// TwinCAT 3 PLC project Strings
// Title: Strings
// Company: _
// Author: Krystian Lis et al.
// ProjectVersion: 1.0.0
// Description: String ops
// ProgramVersion: 3.1.4026.9
// libraries:
//   Tc2_Standard, * (Beckhoff Automation GmbH)
//   Tc2_System, * (Beckhoff Automation GmbH)
//   Tc2_Utilities, * (Beckhoff Automation GmbH)
//   Results, * (_)
// project tree:
//   Strings/Alias/ Ch.TcDUT, Str.TcDUT
//   Strings/SymbolPath/ SymbolPath.TcPOU
//   Strings/Strb/ I_Strb.TcIO, Strb.TcPOU
//   Strings/Strf/ Strf.TcPOU
// (motion and I/O tree: see PLC project broadcast)
// real-time tasks:
//   TASK PlcTask: cycle T#10ms, priority 20, ADS port 350
//   TASK VISU_TASK: cycle T#200000us, priority 30, ADS port 351

// ---- Strings/Alias/Ch.TcDUT
TYPE Ch : STRING(1); END_TYPE

// ---- Strings/Alias/Str.TcDUT
TYPE Str : STRING(255); END_TYPE

// ---- Strings/Strb/I_Strb.TcIO
INTERFACE INTERNAL I_Strb

METHOD Append : I_Strb;
VAR_INPUT
	sToAdd		: Str;
END_VAR
END_METHOD

METHOD FindFirstAfter 	: I_Strb;
VAR_INPUT
	sToFind			: Str;
	nPosition		: INT := 1;
END_VAR
VAR_OUTPUT
	nStart			: INT;
	nEnd			: INT;
END_VAR
END_METHOD

METHOD FindLastBefore 	: I_Strb;
VAR_INPUT
	sToFind			: Str;
	nPosition		: INT := 256;
END_VAR
VAR_OUTPUT
	nStart			: INT;
	nEnd			: INT;
END_VAR
END_METHOD

METHOD HasAfter : BOOL
VAR_INPUT
	sToFind		: Str;
	nPosition	: INT := 0;
END_VAR
VAR_OUTPUT
	nStart			: INT;
	nEnd			: INT;
END_VAR
END_METHOD

METHOD HasBefore : BOOL
VAR_INPUT
	sToFind		: Str;
	nPosition	: INT := 256;
END_VAR
VAR_OUTPUT
	nStart			: INT;
	nEnd			: INT;
END_VAR
END_METHOD

METHOD Inject : I_Strb
VAR_INPUT
	nPosition	: INT;
	sToInject	: Str;
END_VAR
END_METHOD

METHOD IsEmpty : BOOL
VAR_INPUT
END_VAR
END_METHOD

METHOD Length : INT;
VAR_INPUT
END_VAR
END_METHOD

METHOD Prepend : I_Strb;
VAR_INPUT
	sToAdd		: Str;
END_VAR
END_METHOD

METHOD Read : Str;
VAR_INPUT
END_VAR
END_METHOD

METHOD Remove : I_Strb;
VAR_INPUT
	nLength		: INT;
	nPosition	: INT;
END_VAR
END_METHOD

METHOD Set : I_Strb;
VAR_INPUT
	sLiteral	: Str;
END_VAR
END_METHOD

METHOD Slice : I_Strb
VAR_INPUT
	nPosition	: INT;
	nLength		: INT;
END_VAR
VAR_OUTPUT
	sSlice			: Strb;
END_VAR
END_METHOD

METHOD Split : I_Strb;
VAR_INPUT
	nPosition	: INT;
END_VAR
VAR_OUTPUT
	sLeft		: Strb;
	sRight		: Strb;
END_VAR
END_METHOD

END_INTERFACE

// ---- Strings/SymbolPath/SymbolPath.TcPOU
FUNCTION_BLOCK SymbolPath
VAR
	_sPath		: Str;
	_nLen		: INT := 0;
	_nSegStart	: INT := 0;
	_nSegEnd	: INT := 0;
END_VAR

METHOD PRIVATE _HasIncorrectSymbols : BOOL
VAR_INPUT
	sToCheck		: Str;
END_VAR
VAR
	i				: INT;
	_nStrLen		: INT := Tc2_Standard.LEN(sToCheck);
	_sChar			: Ch;
END_VAR
_sChar := Tc2_Standard.MID(sToCheck, 1, 1);
IF (_sChar >= '0') AND (_sChar <= '9') THEN
    _HasIncorrectSymbols := TRUE; // Cannot start with a number
    RETURN;
END_IF;

// Loop through the rest of the string to validate each character
FOR i := 1 TO _nStrLen DO
    _sChar := Tc2_Utilities.F_ToLCase(Tc2_Standard.MID(sToCheck, 1, i));
    
    // Check for invalid characters
    IF NOT ((_sChar >= 'a' AND _sChar <= 'z') OR 	// Lowercase letters
            (_sChar >= '0' AND _sChar <= '9') OR 	// Numbers
            (_sChar = '_') OR                 		// Underscore
			(_sChar = '*')) THEN					// Wildcard
        _HasIncorrectSymbols := TRUE; // Invalid character found
        RETURN;
    END_IF;
END_FOR;

// If no invalid characters are found, return FALSE
_HasIncorrectSymbols := FALSE;
END_METHOD

METHOD AddNext : Results.Result
VAR_INPUT
	sToAdd		: Str;
END_VAR
VAR
	_nNewLen	: INT := _nLen + Tc2_Standard.LEN(sToAdd) + 1;
END_VAR
IF _sPath = '' OR _nSegStart = 0 OR sToAdd = '' THEN
    AddNext := Results.None;
    RETURN;
END_IF;

IF _HasIncorrectSymbols(sToAdd) THEN
	AddNext := Results.None;
	RETURN;
END_IF

IF _nNewLen <= 255 THEN
	_sPath := Tc2_Standard.INSERT(_sPath, '.', _nSegEnd);
	_sPath := Tc2_Standard.INSERT(_sPath, sToAdd, _nSegEnd + 1);
	_nLen := _nNewLen;
	AddNext := Results.Ok;
END_IF
END_METHOD

METHOD AddPrev : Results.Result
VAR_INPUT
	sToAdd		: Str;
END_VAR
VAR
	_nAddLen	: INT := Tc2_Standard.LEN(sToAdd);
	_nNewLen	: INT := _nLen + _nAddLen + 1;
END_VAR
IF _sPath = '' OR _nSegStart = 0 OR sToAdd = '' THEN
    AddPrev := Results.None;
    RETURN;
END_IF;

IF _HasIncorrectSymbols(sToAdd) THEN
	AddPrev := Results.None;
	RETURN;
END_IF

IF _nNewLen <= 255 THEN
	_sPath := Tc2_Standard.INSERT(_sPath, '.', _nSegStart - 1);
	_sPath := Tc2_Standard.INSERT(_sPath, sToAdd, _nSegStart - 2);
	_nLen := _nNewLen;
	_nSegStart := _nSegStart + _nAddLen + 1;
	_nSegEnd := _nSegEnd + _nAddLen + 1;
	AddPrev := Results.Ok;
END_IF
END_METHOD

METHOD Get : Results.Result
VAR_OUTPUT
	sSeg		: Str;
END_VAR
IF _nSegStart = 0 THEN
	RETURN;
END_IF

sSeg := Tc2_Standard.MID(_sPath, _nSegEnd - _nSegStart + 1, _nSegStart);
IF sSeg <> '' THEN
	Get := Results.Ok;
END_IF
END_METHOD

METHOD Next : Results.Result
VAR_OUTPUT
	sSeg		: Str;
END_VAR
VAR
	i			: INT;
END_VAR
// If the path is invalid or already fully processed
IF _sPath = '' OR _nSegEnd = _nLen THEN
    Next := Results.None;
    RETURN;
END_IF;

// Initialize on the first call
IF _nSegStart = 0 THEN
    _nSegStart := 1;
    FOR i := 1 TO _nLen DO
        IF Tc2_Standard.MID(_sPath, 1, i) = '.' THEN
            _nSegEnd := i - 1;
            EXIT;
        END_IF;
    END_FOR;

	IF _nSegEnd < _nSegStart THEN
		_nSegEnd := _nLen;
	END_IF;

    sSeg := Tc2_Standard.MID(_sPath, _nSegEnd - _nSegStart + 1, _nSegStart);
    Next := Results.Ok;
    RETURN;
END_IF;

_nSegStart := _nSegEnd + 2; // Skip the delimiter

FOR i := _nSegStart TO _nLen DO
    IF Tc2_Standard.MID(_sPath, 1, i) = '.' THEN
        _nSegEnd := i - 1;
        EXIT;
    END_IF;
END_FOR;

// If no more delimiters, this is the last segment
IF _nSegEnd < _nSegStart THEN
    _nSegEnd := _nLen;
END_IF;

sSeg := Tc2_Standard.MID(_sPath, _nSegEnd - _nSegStart + 1, _nSegStart);
Next := Results.Ok;
END_METHOD

METHOD Peek : Results.Result
VAR_OUTPUT
	sSeg		: Str;
END_VAR
VAR
	i			: INT;
	_nPeekStart	: INT := 0;
	_nPeekEnd	: INT := 0;
END_VAR
// If the path is invalid or already fully processed
IF _sPath = '' OR _nSegEnd = _nLen OR _nSegStart = 0 THEN
    Peek := Results.None;
    RETURN;
END_IF;

_nPeekStart := _nSegEnd + 2; // Skip the delimiter

FOR i := _nPeekStart TO _nLen DO
    IF Tc2_Standard.MID(_sPath, 1, i) = '.' THEN
        _nPeekEnd := i - 1;
        EXIT;
    END_IF;
END_FOR;

// If no more delimiters, this is the last segment
IF _nPeekEnd = 0 THEN
    _nPeekEnd := _nLen;
END_IF;

sSeg := Tc2_Standard.MID(_sPath, _nPeekEnd - _nPeekStart + 1, _nPeekStart);
Peek := Results.Ok;
END_METHOD

METHOD PeekBack : Results.Result
VAR_OUTPUT
	sSeg		: Str;
END_VAR
VAR
	i			: INT;
	_nPeekStart	: INT := 0;
	_nPeekEnd	: INT := 0;
END_VAR
// If the path is invalid or already fully processed
IF _sPath = '' OR _nSegEnd = 0 OR _nSegStart = 1 THEN
    PeekBack := Results.None;
    RETURN;
END_IF;

_nPeekEnd := _nSegStart - 2; // Skip the delimiter

FOR i := _nPeekEnd TO 1 BY -1 DO
    IF Tc2_Standard.MID(_sPath, 1, i) = '.' THEN
        _nPeekStart := i + 1;
        EXIT;
    END_IF;
END_FOR;

// If no more delimiters, this is the first segment
IF _nPeekStart = 0 THEN
    _nPeekStart := 1;
END_IF;

sSeg := Tc2_Standard.MID(_sPath, _nPeekEnd - _nPeekStart + 1, _nPeekStart);
PeekBack := Results.Ok;
END_METHOD

METHOD Prev : Results.Result
VAR_OUTPUT
	sSeg		: Str;
END_VAR
VAR
	i			: INT;
END_VAR
// If the path is invalid or already fully processed
IF _sPath = '' OR _nSegStart = 1 THEN
    Prev := Results.None;
    RETURN;
END_IF;

// Initialize on the first call
IF _nSegEnd = 0 THEN
    _nSegEnd := _nLen;
    FOR i := _nSegEnd TO 1 BY -1 DO
        IF Tc2_Standard.MID(_sPath, 1, i) = '.' THEN
            _nSegStart := i + 1;
            EXIT;
        END_IF;
    END_FOR;

	// If no more delimiters, this is the first segment
	IF _nSegEnd < _nSegStart THEN
		_nSegStart := 1;
	END_IF;

    sSeg := Tc2_Standard.MID(_sPath, _nSegEnd - _nSegStart + 1, _nSegStart);
    Prev := Results.Ok;
    RETURN;
END_IF;

_nSegEnd := _nSegStart - 2; // Skip the delimiter

FOR i := _nSegEnd TO 1 BY -1 DO
    IF Tc2_Standard.MID(_sPath, 1, i) = '.' THEN
        _nSegStart := i + 1;
        EXIT;
    END_IF;
END_FOR;

// If no more delimiters, this is the first segment
IF _nSegEnd < _nSegStart THEN
    _nSegStart := 1;
END_IF;

sSeg := Tc2_Standard.MID(_sPath, _nSegEnd - _nSegStart + 1, _nSegStart);
Prev := Results.Ok;
END_METHOD

METHOD Read : Str
Read := _sPath;
END_METHOD

METHOD RemoveAndNext : Results.Result
VAR
    _nSegLen		: INT := _nSegEnd - _nSegStart + 1; // Length of the segment to remove
    _bIsFirstSeg	: BOOL := (_nSegStart = 1); // Check if the segment is the first segment
    _bIsLastSeg		: BOOL := (_nSegEnd = _nLen); // Check if the segment is the last segment
	i				: INT;
END_VAR
// Ensure the current path is valid
IF _sPath = '' OR _nSegStart = 0 THEN
    RemoveAndNext := Results.None;
    RETURN;
END_IF;

IF _bIsFirstSeg AND _bIsLastSeg THEN	
	_sPath := '';
    _nLen := 0;
	_nSegStart := 0;
	_nSegEnd := 0;
	RemoveAndNext := Results.Ok;
ELSIF _bIsFirstSeg THEN
	_sPath := Tc2_Standard.DELETE(_sPath, _nSegLen + 1, _nSegStart); // Also removes dot after first segment
	_nLen := _nLen - _nSegLen;
	_nSegStart := 0;
	_nSegEnd := 0;
	RemoveAndNext := Results.Ok;
ELSIF _bIsLastSeg THEN
	_sPath := Tc2_Standard.DELETE(_sPath, _nSegLen + 1, _nSegStart - 1); // Also removes dot before last segment
	_nLen := _nLen - _nSegLen;
	_nSegStart := 0;
	_nSegEnd := 0;
	RemoveAndNext := Results.Ok;
ELSE
	_sPath := Tc2_Standard.DELETE(_sPath, _nSegLen + 1, _nSegStart); // Also removes dot after segment
	_nLen := _nLen - _nSegLen;
	_nSegStart := _nSegEnd + 2; // Skip the delimiter
	
	FOR i := _nSegStart TO _nLen DO
		IF Tc2_Standard.MID(_sPath, 1, i) = '.' THEN
			_nSegEnd := i - 1;
			EXIT;
		END_IF;
	END_FOR;
	
	// If no more delimiters, this is the last segment
	IF _nSegEnd < _nSegStart THEN
		_nSegEnd := _nLen;
	END_IF;
	RemoveAndNext := Results.Ok;
END_IF
END_METHOD

METHOD RemoveAndPrev : Results.Result
VAR
    _nSegLen		: INT := _nSegEnd - _nSegStart + 1; // Length of the segment to remove
    _bIsFirstSeg	: BOOL := (_nSegStart = 1); // Check if the segment is the first segment
    _bIsLastSeg		: BOOL := (_nSegEnd = _nLen); // Check if the segment is the last segment
	i				: INT;
END_VAR
// Ensure the current path is valid
IF _sPath = '' OR _nSegStart = 0 THEN
    RemoveAndPrev := Results.None;
    RETURN;
END_IF;

IF _bIsFirstSeg AND _bIsLastSeg THEN	
	_sPath := '';
    _nLen := 0;
	_nSegStart := 0;
	_nSegEnd := 0;
	RemoveAndPrev := Results.Ok;
ELSIF _bIsFirstSeg THEN
	_sPath := Tc2_Standard.DELETE(_sPath, _nSegLen + 1, _nSegStart); // Also removes dot after first segment
	_nLen := _nLen - _nSegLen;
	_nSegStart := 0;
	_nSegEnd := 0;
	RemoveAndPrev := Results.Ok;
ELSIF _bIsLastSeg THEN
	_sPath := Tc2_Standard.DELETE(_sPath, _nSegLen + 1, _nSegStart - 1); // Also removes dot before last segment
	_nLen := _nLen - _nSegLen;
	_nSegStart := 0;
	_nSegEnd := 0;
	RemoveAndPrev := Results.Ok;
ELSE
	_sPath := Tc2_Standard.DELETE(_sPath, _nSegLen + 1, _nSegStart); // Also removes dot after segment
	_nLen := _nLen - _nSegLen;
	_nSegEnd := _nSegStart - 2; // Skip the delimiter
	
	FOR i := _nSegEnd TO 1 BY -1 DO
		IF Tc2_Standard.MID(_sPath, 1, i) = '.' THEN
			_nSegStart := i + 1;
			EXIT;
		END_IF;
	END_FOR;
	
	// If no more delimiters, this is the first segment
	IF _nSegEnd < _nSegStart THEN
		_nSegStart := 1;
	END_IF;
	RemoveAndPrev := Results.Ok;
END_IF
END_METHOD

METHOD Set : Results.Result
VAR_INPUT
	sNewPath		: Str;
END_VAR
VAR
	i				: INT;
	_nStrLen		: INT := Tc2_Standard.LEN(sNewPath);
	_sChar			: Ch;
END_VAR
IF sNewPath = '' THEN
	RETURN;
END_IF

_sChar := Tc2_Standard.MID(sNewPath, 1, 1);
IF (_sChar >= '0') AND (_sChar <= '9') THEN
    RETURN;
END_IF;

FOR i := 1 TO _nStrLen DO
    _sChar := Tc2_Utilities.F_ToLCase(Tc2_Standard.MID(sNewPath, 1, i));
    
    // Check for invalid characters
    IF NOT ((_sChar >= 'a' AND _sChar <= 'z') OR 	// Lowercase letters
            (_sChar >= '0' AND _sChar <= '9') OR 	// Numbers
            (_sChar = '_') OR                 		// Underscore
			(_sChar = '.') OR
			(_sChar = '*')) THEN					// Wildcard
        RETURN;
    END_IF;
END_FOR;

IF Tc2_Standard.FIND(sNewPath, '..') <> 0 THEN
	RETURN;
END_IF

IF Tc2_Standard.FIND(sNewPath, '**') <> 0 THEN
	RETURN;
END_IF

_sPath := sNewPath;
_nLen := _nStrLen;
END_METHOD

METHOD Swap : Results.Result
VAR_INPUT
	sToSwap		: Str;
END_VAR
VAR
	_nSegLen	: INT := _nSegEnd - _nSegStart + 1;
	_nSwapLen	: INT := Tc2_Standard.LEN(sToSwap);
	_nNewLen	: INT := _nLen - _nSegLen + _nSwapLen;
END_VAR
IF _sPath = '' OR _nSegStart = 0 OR sToSwap = '' THEN
    Swap := Results.None;
    RETURN;
END_IF;

IF _HasIncorrectSymbols(sToSwap) THEN
	Swap := Results.None;
	RETURN;
END_IF

IF _nNewLen <= 255 THEN
	_sPath := Tc2_Standard.REPLACE(_sPath, sToSwap, _nSegLen, _nSegStart);
	_nSegEnd := _nSegStart + _nSwapLen - 1;
	_nLen := _nNewLen;
	Swap := Results.Ok;
END_IF
END_METHOD

END_FUNCTION_BLOCK

// ---- Strings/Strb/Strb.TcPOU
FUNCTION_BLOCK Strb IMPLEMENTS I_Strb
VAR
	_sString	: Str;
	_nLength	: INT;
END_VAR

PROPERTY PRIVATE _this : I_Strb
GET
VAR
	_iThis : I_Strb := THIS^;
END_VAR
_this := _iThis;
END_GET
END_PROPERTY

METHOD Append : I_Strb;
VAR_INPUT
	sToAdd		: Str;
END_VAR
VAR
	_nNewLength	: INT;
END_VAR
Append := _this;

IF sToAdd = '' THEN
	RETURN;
END_IF

_nNewLength := Tc2_Standard.LEN(sToAdd) + _nLength;
IF _nNewLength > 255 THEN
	_nNewLength := 255;
END_IF

_sString := Tc2_Standard.CONCAT(_sString, sToAdd);
_nLength := _nNewLength;
END_METHOD

METHOD FindFirstAfter 	: I_Strb;
VAR_INPUT
	sToFind			: Str;
	nPosition		: INT := 1;
END_VAR
VAR_OUTPUT
	nStart			: INT;
	nEnd			: INT;
END_VAR
VAR
	_sTemp			: Str;
	_nOffset		: INT;
END_VAR
FindFirstAfter := _this;

IF sToFind = '' THEN
	RETURN;
END_IF

IF nPosition = 0 THEN
	RETURN;
END_IF

_sTemp := Tc2_Standard.MID(_sString, _nLength, nPosition);
IF (_nOffset := Tc2_Standard.FIND(_sTemp, sToFind)) <> 0 THEN
	nStart := nPosition + _nOffset - 1;
	nEnd := nPosition + _nOffset - 2 + Tc2_Standard.LEN(sToFind);
END_IF
END_METHOD

METHOD FindLastBefore 	: I_Strb;
VAR_INPUT
	sToFind			: Str;
	nPosition		: INT := 256;
END_VAR
VAR_OUTPUT
	nStart			: INT;
	nEnd			: INT;
END_VAR
VAR
	_sTemp			: Str;
	_nFindLength	: INT := Tc2_Standard.LEN(sToFind);
	_nOffset		: INT;
END_VAR
FindLastBefore := _this;

IF sToFind = '' THEN
	RETURN;
END_IF

IF nPosition = 0 THEN
	RETURN;
END_IF

IF nPosition = 256 THEN
	nPosition := _nLength;
END_IF

REPEAT
	_sTemp := Tc2_Standard.MID(_sString, _nFindLength, nPosition);
	IF _sTemp = sToFind THEN
		nStart 	:= nPosition;
		nEnd	:= nPosition + _nFindLength - 1;
		RETURN;
	END_IF
UNTIL
	(nPosition := nPosition - 1) <= 0
END_REPEAT
END_METHOD

METHOD HasAfter : BOOL
VAR_INPUT
	sToFind		: Str;
	nPosition	: INT := 0;
END_VAR
VAR_OUTPUT
	nStart			: INT;
	nEnd			: INT;
END_VAR
FindFirstAfter(sToFind, nPosition, nStart => nStart, nEnd => nEnd);
HasAfter := nStart > 0;
END_METHOD

METHOD HasBefore : BOOL
VAR_INPUT
	sToFind		: Str;
	nPosition	: INT := 256;
END_VAR
VAR_OUTPUT
	nStart			: INT;
	nEnd			: INT;
END_VAR
IF nPosition = 256 THEN
	nPosition := Tc2_Standard.LEN(_sString);
END_IF

FindLastBefore(sToFind, nPosition, nStart => nStart, nEnd => nEnd);
HasBefore := nStart > 0;
END_METHOD

METHOD Inject : I_Strb
VAR_INPUT
	nPosition	: INT;
	sToInject	: Str;
END_VAR
VAR
	_nNewLength	: INT;
END_VAR
Inject := _this;

IF sToInject = '' THEN
	RETURN;
END_IF

IF nPosition = 0 THEN
	RETURN;
END_IF

IF nPosition > _nLength THEN
	RETURN;
END_IF

_nNewLength := Tc2_Standard.LEN(sToInject) + _nLength;
IF _nNewLength > 255 THEN
	_nNewLength := 255;
END_IF

_sString := Tc2_Standard.INSERT(_sString, sToInject, nPosition);
_nLength := _nNewLength;
END_METHOD

METHOD IsEmpty : BOOL
VAR_INPUT
END_VAR
IsEmpty := _nLength = 0;
END_METHOD

METHOD Length : INT;
VAR_INPUT
END_VAR
Length := _nLength;
END_METHOD

METHOD Prepend : I_Strb;
VAR_INPUT
	sToAdd		: Str;
END_VAR
VAR
	_nNewLength	: INT;
END_VAR
Prepend := _this;

IF sToAdd = '' THEN
	RETURN;
END_IF

_nNewLength := Tc2_Standard.LEN(sToAdd) + _nLength;
IF _nNewLength > 255 THEN
	_nNewLength := 255;
END_IF

_sString := Tc2_Standard.CONCAT(sToAdd, _sString);
_nLength := _nNewLength;
END_METHOD

METHOD Read : Str;
VAR_INPUT
END_VAR
Read := _sString;
END_METHOD

METHOD Remove : I_Strb;
VAR_INPUT
	nLength		: INT;
	nPosition	: INT;
END_VAR
VAR
	_nPosition	: INT;
END_VAR
Remove := _this;

IF nPosition = 0 THEN
	RETURN;
END_IF

IF nPosition > _nLength THEN
	RETURN;
END_IF

IF nLength = 0 THEN
	RETURN;
END_IF

IF nLength + nPosition > _nLength THEN
	nLength := _nLength - nPosition + 1;
END_IF

_sString := Tc2_Standard.DELETE(_sString, nLength, nPosition);
_nLength := _nLength - nLength;
END_METHOD

METHOD Set : I_Strb;
VAR_INPUT
	sLiteral	: Str;
END_VAR
Set 		:= _this;

_sString 	:= sLiteral;
_nLength	:= Tc2_Standard.LEN(sLiteral);
END_METHOD

METHOD Slice : I_Strb
VAR_INPUT
	nPosition	: INT;
	nLength		: INT;
END_VAR
VAR_OUTPUT
	sSlice			: Strb;
END_VAR
Slice := _this;

IF nPosition = 0 THEN
	RETURN;
END_IF

IF nLength = 0 THEN
	RETURN;
END_IF

sSlice.Set(Tc2_Standard.MID(_sString, nLength, nPosition));
END_METHOD

METHOD Split : I_Strb;
VAR_INPUT
	nPosition	: INT;
END_VAR
VAR_OUTPUT
	sLeft		: Strb;
	sRight		: Strb;
END_VAR
Split := _this;

IF nPosition = 0 THEN
	RETURN;
END_IF

sLeft.Set(Tc2_Standard.LEFT(_sString, nPosition));
sRight.Set(Tc2_Standard.RIGHT(_sString, _nLength - nPosition));
END_METHOD

END_FUNCTION_BLOCK

// ---- Strings/Strf/Strf.TcPOU
PROGRAM Strf

METHOD Float					: Str;
VAR_INPUT
	rValue						: ANY_REAL;	

	nTrailingZeroes				: USINT := 0;
	nLeadingZeroes				: USINT := 0;
END_VAR
VAR
	_rReal						: REAL;
	_rLReal						: LREAL;
	_sBase						: Strb;
	_nDotPos					: INT;
	_Resulteger					: Strb;
	_sFraction					: Strb;
END_VAR
CASE rValue.TypeClass OF
	__SYSTEM.TYPE_CLASS.TYPE_REAL:
		Tc2_System.MEMMOVE(ADR(_rReal), rValue.pValue, DINT_TO_UDINT(rValue.diSize));
		_rLReal := REAL_TO_LREAL(_rReal);
		
	__SYSTEM.TYPE_CLASS.TYPE_LREAL:
		Tc2_System.MEMMOVE(ADR(_rLReal), rValue.pValue, DINT_TO_UDINT(rValue.diSize));
END_CASE

_sBase.Set(LREAL_TO_STRING(_rLReal))
		.FindFirstAfter('.', 1, nStart => _nDotPos)
		.Split(_nDotPos, sLeft => _Resulteger, sRight => _sFraction);

_sFraction.Slice(1, nTrailingZeroes, sSlice => _sFraction)
				.Set(Padding(_sFraction.Read(), 0, nTrailingZeroes, '0'));
				
_Resulteger.Remove(1, _Resulteger.Length())
				.Set(Padding(_Resulteger.Read(), nLeadingZeroes, 0, '0'))
				.Append('.')
				.Append(_sFraction.Read());

Float := _Resulteger.Read();
END_METHOD

METHOD Integer : Str
VAR_INPUT
	nValue			: ANY_INT;
	nLeadingZeroes	: USINT := 0;
END_VAR
VAR
	_nSigned		: LINT;
	_nUnsigned		: ULINT;
END_VAR
CASE nValue.TypeClass OF
	__SYSTEM.TYPE_CLASS.TYPE_SINT,
	__SYSTEM.TYPE_CLASS.TYPE_INT,
	__SYSTEM.TYPE_CLASS.TYPE_DINT,
	__SYSTEM.TYPE_CLASS.TYPE_LINT:
		Tc2_System.MEMMOVE(ADR(_nSigned), nValue.pValue, DINT_TO_UDINT(nValue.diSize));
		Integer := Padding(LINT_TO_STRING(_nSigned), nLeadingZeroes, 0, '0');
		
	__SYSTEM.TYPE_CLASS.TYPE_USINT,
	__SYSTEM.TYPE_CLASS.TYPE_UINT,
	__SYSTEM.TYPE_CLASS.TYPE_UDINT,
	__SYSTEM.TYPE_CLASS.TYPE_ULINT:	
		Tc2_System.MEMMOVE(ADR(_nUnsigned), nValue.pValue, DINT_TO_UDINT(nValue.diSize));
		Integer := Padding(ULINT_TO_STRING(_nUnsigned), nLeadingZeroes, 0, '0');
END_CASE
END_METHOD

METHOD Padding				: Str;
VAR_INPUT
	sValue					: Str;
	nLeftPadding			: USINT := 0;
	nRightPadding			: USINT := 0;
	sFillChar				: Ch	:= ' ';
END_VAR
VAR
	_sBase					: Strb;
	_sLeft					: Strb;
	_sRight					: Strb;
END_VAR
_sBase.Set(sValue);
IF nRightPadding = 0 THEN
	WHILE _sBase.Length() < nLeftPadding DO
		_sBase.Prepend(sFillChar);
	END_WHILE
ELSIF nLeftPadding = 0 THEN
	WHILE _sBase.Length() < nRightPadding DO
		_sBase.Append(sFillChar);
	END_WHILE
ELSE
	_sBase.Split(_sBase.Length()/2, sLeft => _sLeft, sRight => _sRight);
	WHILE _sLeft.Length() < nLeftPadding DO
		_sLeft.Prepend(sFillChar);
	END_WHILE
	WHILE _sRight.Length() < nRightPadding DO
		_sRight.Append(sFillChar);
	END_WHILE
	
	_sLeft.Append(_sRight.Read());
	_sBase.Set(_sLeft.Read());
END_IF

Padding := _sBase.Read();
END_METHOD

METHOD SimpleTime : Str
VAR_INPUT
	tValue		: TIME;
	sMinUnit	: Str := 'MS'; //Possible options: MS, S, M, H, D
	sMaxUnit	: Str := 'S'; //Possible options: MS, S, M, H, D
END_VAR
VAR
	_nMinUnit	: USINT;
	_nMaxUnit	: USINT;
	_sValues	: ARRAY[1..5] OF Strb;
	_nValues	: ARRAY[1..5] OF UINT;
	_sUnits   	: ARRAY[1..5] OF STRING := ['MS', 'S', 'M', 'H', 'D'];
	_stTime		: Tc2_Utilities.OTSTRUCT;
	_i			: USINT;
	_strb		: Strb;
END_VAR
FOR _i := 1 TO 5 DO
	IF _sUnits[_i] = sMinUnit THEN
		_nMinUnit := _i;
	END_IF
	IF _sUnits[_i] = sMaxUnit THEN
		_nMaxUnit := _i;
	END_IF
END_FOR

IF _nMaxUnit = 0 THEN
	RETURN;
END_IF

IF _nMinUnit = 0 THEN
	RETURN;
END_IF

IF _nMinUnit > _nMaxUnit THEN
	RETURN;
END_IF

_stTime := Tc2_Utilities.TIME_TO_OTSTRUCT(tValue);
_stTime.wDay := _stTime.wWeek * 7 + _stTime.wDay;

_nValues[1] := WORD_TO_UINT(_stTime.wMilliseconds);
_nValues[2] := WORD_TO_UINT(_stTime.wSecond);
_nValues[3] := WORD_TO_UINT(_stTime.wMinute);
_nValues[4] := WORD_TO_UINT(_stTime.wHour);
_nValues[5] := WORD_TO_UINT(_stTime.wDay);

_sValues[1].Set(Strf.Integer(_nValues[1], 3)).Append('ms');
_sValues[2].Set(Strf.Integer(_nValues[2], 2)).Append('s');
_sValues[3].Set(Strf.Integer(_nValues[3], 2)).Append('m');
_sValues[4].Set(Strf.Integer(_nValues[4], 2)).Append('h');
_sValues[5].Set(Strf.Integer(_nValues[5], 3)).Append('d');

IF _nMaxUnit < 5 THEN
    FOR _i := 5 TO _nMaxUnit + 1 BY -1 DO
        IF _nValues[_i] <> 0 THEN
            _strb.Append(_sValues[_i].Read()).Append(' ');
        END_IF
    END_FOR
END_IF

FOR _i := _nMaxUnit TO _nMinUnit BY -1 DO
    _strb.Append(_sValues[_i].Read()).Append(' ');
END_FOR

SimpleTime := _strb.Read();
END_METHOD

END_PROGRAM
